// Library/POUs/ForceControl/MC_ReadActualForce/Structures/ReadActualForceSendData
{attribute 'pack_mode' := '1'}
// ------------------------------------------------------------------------- 
//  SRCI Robot Library                                                
// ------------------------------------------------------------------------- 
//                                                                           
//  Object:      ReadActualForceSendData                                       
//  Author:      Thorsten Brach                                                
//  Date:        2024-06-11
//
//  Description:                                              
//   
//                                                                           
//  Copyright: 
//    (C) 2024 Thorsten Brach. All rights reserved                                                                                                                                            
//             Licensed under the LGPL-3.0 license.
//                                                                           
//  Disclaimer:                                                                           
//    This project is provided without any guarantee and can be used for   
//    private and commercial purposes. Any use is at the user’s 
//    own risk and responsibility.
//
// -------------------------------------------------------------------------
TYPE ReadActualForceSendData EXTENDS CmdHeader:   
STRUCT
  /// ID of Action that will be executed when this command is active
  /// • >0: Start Action        - Start executing the Action function with the identical ListenerID.
  /// • <0: Stop Action         - Stop executing the Action function with the identical ListenerID.
  /// •  0: Undefined (default) - If no EmitterID is defined, the function returns an error message
  /// For more information see chapter 5.5.12.4
  EmitterID          : ARRAY [0..3] OF SINT;
  /// ListenerID
  ListenerID         : SINT; 
  /// Reserve
  Reserve            : BYTE; 
  /// Index of tool
  /// •      0: Flange (default)
  /// • 1..254: Tool frames
  ToolNo             : USINT;
  /// Define the index number of the UCS that will be assigned to the conveyor.
  /// For more information refer to chapter 5.5.14
  FrameNo            : USINT;
  /// Index of payload data containing mass, center of gravity, orientation and inertia relative to SensorFrame.
  /// Required to calibrate system for setting up gravity compensation and sensor offset.
  CalibrationData    : USINT;
  /// Defines type of reference of Force and Torque (at least one option must be supported )
  ReferenceType      : ReferenceType;
END_STRUCT
END_TYPE

// Library/POUs/General/MC_EnableRobot/Structures/EnableRobotOutCmd
{attribute 'pack_mode' := '1'} 
// ------------------------------------------------------------------------- 
//  SRCI Robot Library                                                
// ------------------------------------------------------------------------- 
//                                                                           
//  Object:      EnableRobotOutCmd                                       
//  Author:      Thorsten Brach                                                
//  Date:        2024-06-01
//
//  Description:                                              
//   
//                                                                           
//  Copyright: 
//    (C) 2024 Thorsten Brach. All rights reserved                                                                                                                                            
//             Licensed under the LGPL-3.0 license.
//                                                                           
//  Disclaimer:                                                                           
//    This project is provided without any guarantee and can be used for   
//    private and commercial purposes. Any use is at the user’s 
//    own risk and responsibility.
//
// -------------------------------------------------------------------------
TYPE EnableRobotOutCmd :
STRUCT
END_STRUCT
END_TYPE

// Library/POUs/General/MC_EnableRobot/Structures/EnableRobotParCmd
{attribute 'pack_mode' := '1'} 
// ------------------------------------------------------------------------- 
//  SRCI Robot Library                                                
// ------------------------------------------------------------------------- 
//                                                                           
//  Object:      EnableRobotParCmd                                       
//  Author:      Thorsten Brach                                                
//  Date:        2024-06-01
//
//  Description:                                              
//   
//                                                                           
//  Copyright: 
//    (C) 2024 Thorsten Brach. All rights reserved                                                                                                                                            
//             Licensed under the LGPL-3.0 license.
//                                                                           
//  Disclaimer:                                                                           
//    This project is provided without any guarantee and can be used for   
//    private and commercial purposes. Any use is at the user’s 
//    own risk and responsibility.
//
// -------------------------------------------------------------------------
TYPE EnableRobotParCmd :
STRUCT
  /// The robot will move while HoldToRun is set TRUE
  HoldToRun  : BOOL;
  /// While activated the RI state switches to interrupted when a buffered command returns Done TRUE
  /// At least one of the optional modes must be supported
  StepMode   : StepMode;
  /// Relates to StepMode 1 (Blending) and 2 (Exact stop)
  /// Start the next buffered command with the rising edge in T1 External or T2 External
  ManualStep : BOOL;  
END_STRUCT
END_TYPE

// Library/POUs/General/MC_EnableRobot/Structures/EnableRobotRecvData
{attribute 'pack_mode' := '1'} 
// ------------------------------------------------------------------------- 
//  SRCI Robot Library                                                
// ------------------------------------------------------------------------- 
//                                                                           
//  Object:      EnableRobotRecvData                                       
//  Author:      Thorsten Brach                                                
//  Date:        2024-06-01
//
//  Description:                                              
//   
//                                                                           
//  Copyright: 
//    (C) 2024 Thorsten Brach. All rights reserved                                                                                                                                            
//             Licensed under the LGPL-3.0 license.
//                                                                           
//  Disclaimer:                                                                           
//    This project is provided without any guarantee and can be used for   
//    private and commercial purposes. Any use is at the user’s 
//    own risk and responsibility.
//
// -------------------------------------------------------------------------
TYPE EnableRobotRecvData EXTENDS RspHeader :
STRUCT
  /// TRUE when robot is set to RA power state "Enabled".
  Enabled : BOOL;
END_STRUCT
END_TYPE

// Library/POUs/General/MC_EnableRobot/Structures/EnableRobotSendData
{attribute 'pack_mode' := '1'}
// ------------------------------------------------------------------------- 
//  SRCI Robot Library                                                
// ------------------------------------------------------------------------- 
//                                                                           
//  Object:      ActivateNextCommandParCmd                                       
//  Author:      Thorsten Brach                                                
//  Date:        2024-06-01
//
//  Description:                                              
//   
//                                                                           
//  Copyright: 
//    (C) 2024 Thorsten Brach. All rights reserved                                                                                                                                            
//             Licensed under the LGPL-3.0 license.
//                                                                           
//  Disclaimer:                                                                           
//    This project is provided without any guarantee and can be used for   
//    private and commercial purposes. Any use is at the user’s 
//    own risk and responsibility.
//
// -------------------------------------------------------------------------
TYPE EnableRobotSendData EXTENDS CmdHeader: 
STRUCT
  /// Set TRUE to change RA power state to "Enabled"
 Enable          : BOOL;
 /// The robot will move while HoldToRun is set TRUE
 HoldToRun       : BOOL;
 /// While activated the RI state switches to interrupted when a buffered command returns Done TRUE
 /// At least one of the optional modes must be supported
 StepMode        : StepMode;
 /// Relates to StepMode 1 (Blending) and 2 (Exact stop)
 /// Start the next buffered command with the rising edge in T1 External or T2 External
 ManualStep      : BOOL;  
END_STRUCT
END_TYPE

// Library/POUs/General/MC_GroupReset/Structures/GroupResetOutCmd
{attribute 'pack_mode' := '1'} 
// ------------------------------------------------------------------------- 
//  SRCI Robot Library                                                
// ------------------------------------------------------------------------- 
//                                                                           
//  Object:      GroupResetOutCmd                                       
//  Author:      Thorsten Brach                                                
//  Date:        2024-06-17
//
//  Description:                                              
//   
//                                                                           
//  Copyright: 
//    (C) 2024 Thorsten Brach. All rights reserved                                                                                                                                            
//             Licensed under the LGPL-3.0 license.
//                                                                           
//  Disclaimer:                                                                           
//    This project is provided without any guarantee and can be used for   
//    private and commercial purposes. Any use is at the user’s 
//    own risk and responsibility.
//
// -------------------------------------------------------------------------
TYPE GroupResetOutCmd :
STRUCT
END_STRUCT
END_TYPE

// Library/POUs/General/MC_GroupReset/Structures/GroupResetParCmd
{attribute 'pack_mode' := '1'} 
// ------------------------------------------------------------------------- 
//  SRCI Robot Library                                                
// ------------------------------------------------------------------------- 
//                                                                           
//  Object:      GroupResetParCmd                                       
//  Author:      Thorsten Brach                                                
//  Date:        2024-06-17
//
//  Description:                                              
//   
//                                                                           
//  Copyright: 
//    (C) 2024 Thorsten Brach. All rights reserved                                                                                                                                            
//             Licensed under the LGPL-3.0 license.
//                                                                           
//  Disclaimer:                                                                           
//    This project is provided without any guarantee and can be used for   
//    private and commercial purposes. Any use is at the user’s 
//    own risk and responsibility.
//
// -------------------------------------------------------------------------
TYPE GroupResetParCmd :
STRUCT
END_STRUCT
END_TYPE

// Library/POUs/General/MC_GroupReset/Structures/GroupResetRecvData
{attribute 'pack_mode' := '1'} 
// ------------------------------------------------------------------------- 
//  SRCI Robot Library                                                
// ------------------------------------------------------------------------- 
//                                                                           
//  Object:      GroupResetRecvData                                       
//  Author:      Thorsten Brach                                                
//  Date:        2024-06-17
//
//  Description:                                              
//   
//                                                                           
//  Copyright: 
//    (C) 2024 Thorsten Brach. All rights reserved                                                                                                                                            
//             Licensed under the LGPL-3.0 license.
//                                                                           
//  Disclaimer:                                                                           
//    This project is provided without any guarantee and can be used for   
//    private and commercial purposes. Any use is at the user’s 
//    own risk and responsibility.
//
// -------------------------------------------------------------------------
TYPE GroupResetRecvData EXTENDS RspHeader :
STRUCT
END_STRUCT
END_TYPE

// Library/POUs/General/MC_GroupReset/Structures/GroupResetSendData
{attribute 'pack_mode' := '1'}
// ------------------------------------------------------------------------- 
//  SRCI Robot Library                                                
// ------------------------------------------------------------------------- 
//                                                                           
//  Object:      GroupResetSendData                                       
//  Author:      Thorsten Brach                                                
//  Date:        2024-06-17
//
//  Description:                                              
//   
//                                                                           
//  Copyright: 
//    (C) 2024 Thorsten Brach. All rights reserved                                                                                                                                            
//             Licensed under the LGPL-3.0 license.
//                                                                           
//  Disclaimer:                                                                           
//    This project is provided without any guarantee and can be used for   
//    private and commercial purposes. Any use is at the user’s 
//    own risk and responsibility.
//
// -------------------------------------------------------------------------
TYPE GroupResetSendData EXTENDS CmdHeader:   
STRUCT
END_STRUCT
END_TYPE

// Library/POUs/General/MC_RestartController/Structures/RestartControllerOutCmd
{attribute 'pack_mode' := '1'} 
// ------------------------------------------------------------------------- 
//  SRCI Robot Library                                                
// ------------------------------------------------------------------------- 
//                                                                           
//  Object:      RestartControllerOutCmd                                       
//  Author:      Thorsten Brach                                                
//  Date:        2024-06-22
//
//  Description:                                              
//   
//                                                                           
//  Copyright: 
//    (C) 2024 Thorsten Brach. All rights reserved                                                                                                                                            
//             Licensed under the LGPL-3.0 license.
//                                                                           
//  Disclaimer:                                                                           
//    This project is provided without any guarantee and can be used for   
//    private and commercial purposes. Any use is at the user’s 
//    own risk and responsibility.
//
// -------------------------------------------------------------------------
TYPE RestartControllerOutCmd :
STRUCT
  /// TRUE when execution of command has been confirmed by RC and restart is about to be initiated.
  RestartAccepted : BOOL;  
END_STRUCT
END_TYPE

// Library/POUs/General/MC_RestartController/Structures/RestartControllerParCmd
{attribute 'pack_mode' := '1'} 
// ------------------------------------------------------------------------- 
//  SRCI Robot Library                                                
// ------------------------------------------------------------------------- 
//                                                                           
//  Object:      RestartControllerParCmd                                       
//  Author:      Thorsten Brach                                                
//  Date:        2024-06-22
//
//  Description:                                              
//   
//                                                                           
//  Copyright: 
//    (C) 2024 Thorsten Brach. All rights reserved                                                                                                                                            
//             Licensed under the LGPL-3.0 license.
//                                                                           
//  Disclaimer:                                                                           
//    This project is provided without any guarantee and can be used for   
//    private and commercial purposes. Any use is at the user’s 
//    own risk and responsibility.
//
// -------------------------------------------------------------------------
TYPE RestartControllerParCmd :
STRUCT
END_STRUCT
END_TYPE

// Library/POUs/General/MC_RestartController/Structures/RestartControllerRecvData
{attribute 'pack_mode' := '1'} 
// ------------------------------------------------------------------------- 
//  SRCI Robot Library                                                
// ------------------------------------------------------------------------- 
//                                                                           
//  Object:      RestartControllerRecvData                                       
//  Author:      Thorsten Brach                                                
//  Date:        2024-06-22
//
//  Description:                                              
//   
//                                                                           
//  Copyright: 
//    (C) 2024 Thorsten Brach. All rights reserved                                                                                                                                            
//             Licensed under the LGPL-3.0 license.
//                                                                           
//  Disclaimer:                                                                           
//    This project is provided without any guarantee and can be used for   
//    private and commercial purposes. Any use is at the user’s 
//    own risk and responsibility.
//
// -------------------------------------------------------------------------
TYPE RestartControllerRecvData EXTENDS RspHeader :
STRUCT
  /// TRUE when execution of command has been confirmed by RC and restart is about to be initiated.
  RestartAccepted : BOOL;
END_STRUCT
END_TYPE

// Library/POUs/General/MC_RestartController/Structures/RestartControllerSendData
{attribute 'pack_mode' := '1'}
// ------------------------------------------------------------------------- 
//  SRCI Robot Library                                                
// ------------------------------------------------------------------------- 
//                                                                           
//  Object:      RestartControllerSendData                                       
//  Author:      Thorsten Brach                                                
//  Date:        2024-06-22
//
//  Description:                                              
//   
//                                                                           
//  Copyright: 
//    (C) 2024 Thorsten Brach. All rights reserved                                                                                                                                            
//             Licensed under the LGPL-3.0 license.
//                                                                           
//  Disclaimer:                                                                           
//    This project is provided without any guarantee and can be used for   
//    private and commercial purposes. Any use is at the user’s 
//    own risk and responsibility.
//
// -------------------------------------------------------------------------
TYPE RestartControllerSendData EXTENDS CmdHeader: 
STRUCT
END_STRUCT
END_TYPE

// Library/POUs/General/MC_RobotTask/Structures/ParCfg/Com/RobotTaskParCfgCom
{attribute 'pack_mode' := '1'} 
// ------------------------------------------------------------------------- 
//  SRCI Robot Library                                                
// ------------------------------------------------------------------------- 
//                                                                           
//  Object:      RobotTaskParCfgCom                                       
//  Author:      Thorsten Brach                                                
//  Date:        2024-11-30
//
//  Description:                                              
//   
//                                                                           
//  Copyright: 
//    (C) 2024 Thorsten Brach. All rights reserved                                                                                                                                            
//             Licensed under the LGPL-3.0 license.
//                                                                           
//  Disclaimer:                                                                           
//    This project is provided without any guarantee and can be used for   
//    private and commercial purposes. Any use is at the user’s 
//    own risk and responsibility.
//
// -------------------------------------------------------------------------
TYPE RobotTaskParCfgCom :
STRUCT
  /// Maximum allowed time between incrementation of LifeSign before communication error.
  /// • <10 ms: Invalid
  /// • 50 ms: default
  /// See also chapter 5.6.6.2.
  LifeSignTimeOut        : TIME := T#50MS;
  /// Number of Bytes of the frame to be used for the telegram of the given Axisgroup. Direction client to server
  TelegramLengthPlcToRob : UINT := 256;
  /// Number of Bytes of the frame to be used for the telegram of the given Axisgroup. Direction server to client
  TelegramLengthRobToPlc : UINT := 256;  
END_STRUCT
END_TYPE

// Library/POUs/General/MC_RobotTask/Structures/ParCfg/Plc/RobotTaskParCfgPlc
{attribute 'pack_mode' := '1'} 
// ------------------------------------------------------------------------- 
//  SRCI Robot Library                                                
// ------------------------------------------------------------------------- 
//                                                                           
//  Object:      RobotTaskParCfgPlc                                       
//  Author:      Thorsten Brach                                                
//  Date:        2024-11-30
//
//  Description:                                              
//   
//                                                                           
//  Copyright: 
//    (C) 2024 Thorsten Brach. All rights reserved                                                                                                                                            
//             Licensed under the LGPL-3.0 license.
//                                                                           
//  Disclaimer:                                                                           
//    This project is provided without any guarantee and can be used for   
//    private and commercial purposes. Any use is at the user’s 
//    own risk and responsibility.
//
// -------------------------------------------------------------------------
TYPE RobotTaskParCfgPlc :
STRUCT
  /// PLC cycle time
  CycleTime           : TIME := T#10MS;
  /// parameter
  Parameter           : RobotTaskParCfgPlcParameter;  
  /// Configuration of optional cyclic data send to the Robot
  OptionalCyclic      : AxesGroupParameterPlcOptionalCyclic; {warning 'Remove - this is already part of RobotTaskParCfgPlcParameter'}
END_STRUCT
END_TYPE

// Library/POUs/General/MC_RobotTask/Structures/ParCfg/Plc/RobotTaskParCfgPlcParameter
{attribute 'pack_mode' := '1'} 
// ------------------------------------------------------------------------- 
//  SRCI Robot Library                                                
// ------------------------------------------------------------------------- 
//                                                                           
//  Object:      RobotTaskParCfgPlcParameter                                       
//  Author:      Thorsten Brach                                                
//  Date:        2024-11-30
//
//  Description:                                              
//   
//                                                                           
//  Copyright: 
//    (C) 2024 Thorsten Brach. All rights reserved                                                                                                                                            
//             Licensed under the LGPL-3.0 license.
//                                                                           
//  Disclaimer:                                                                           
//    This project is provided without any guarantee and can be used for   
//    private and commercial purposes. Any use is at the user’s 
//    own risk and responsibility.
//
// -------------------------------------------------------------------------
TYPE RobotTaskParCfgPlcParameter EXTENDS AxesGroupParameterPlcParameter :
STRUCT
END_STRUCT
END_TYPE

// Library/POUs/General/MC_RobotTask/Structures/ParCfg/Rob/RobotTaskParCfgRob
TYPE RobotTaskParCfgRob :
STRUCT
// ------------------------------------------------------------------------- 
//  SRCI Robot Library                                                
// ------------------------------------------------------------------------- 
//                                                                           
//  Object:      RobotTaskParCfgRob                                       
//  Author:      Thorsten Brach                                                
//  Date:        2024-11-30
//
//  Description:                                              
//   
//                                                                           
//  Copyright: 
//    (C) 2024 Thorsten Brach. All rights reserved                                                                                                                                            
//             Licensed under the LGPL-3.0 license.
//                                                                           
//  Disclaimer:                                                                           
//    This project is provided without any guarantee and can be used for   
//    private and commercial purposes. Any use is at the user’s 
//    own risk and responsibility.
//
// -------------------------------------------------------------------------
  /// Robot parameter
  Parameter      : RobotTaskParCfgRobParameter;
  /// Configuration of optional cyclic data received from the Robot
  OptionalCyclic : AxesGroupParameterRobOptionalCyclic;
END_STRUCT
END_TYPE

// Library/POUs/General/MC_RobotTask/Structures/ParCfg/Rob/RobotTaskParCfgRobParameter
{attribute 'pack_mode' := '1'} 
// ------------------------------------------------------------------------- 
//  SRCI Robot Library                                                
// ------------------------------------------------------------------------- 
//                                                                           
//  Object:      RobotTaskParCfgRobParameter                                       
//  Author:      Thorsten Brach                                                
//  Date:        2024-11-30
//
//  Description:                                              
//   
//                                                                           
//  Copyright: 
//    (C) 2024 Thorsten Brach. All rights reserved                                                                                                                                            
//             Licensed under the LGPL-3.0 license.
//                                                                           
//  Disclaimer:                                                                           
//    This project is provided without any guarantee and can be used for   
//    private and commercial purposes. Any use is at the user’s 
//    own risk and responsibility.
//
// -------------------------------------------------------------------------
TYPE RobotTaskParCfgRobParameter :
STRUCT
  /// Defines blending behavior for single move commands. One of the optional modes must be supported.
  ///  • 0 (default): Move to end position
  ///       Robot moves exactly the target position independently of the selected "BlendingMode"
  ///  • 1: Wait at blending parameter 
  ///       Robot stops its movement when the specified blending parameter is reached
  WaitAtBlendingZone         : BOOL;
  /// Allow a sequence switch from primary to secondary while a subprogram called via CallSubprogram (6.5.18) in the sequence is in progress
  AllowSecSeqWhileSubprogram : BOOL;
  /// Allows blending when CallSubprogram is called in sequence and removed afterwards. For more information see chapter 6.5.21.
  /// • 0 (default): Dynamic blending is prevented
  /// • 1: Dynamic blending is allowed
  AllowDynamicBlending       : BOOL;
  /// Defines waiting time of RC between receiving a first move command when motion queue is empty and starting the first movement. See also chapter 5.6.8.
  DelayTime                  : UINT;
  /// Define number of points required to calculate the blending. See also chapter 5.6.8.
  WaitForNrOfCmd             : UINT;
  /// Defines a delay time between detecting an inconsistency of configuration data between server and client and executing the defined SyncReaction. 
  /// Always positive. Default: 0 ms
  SyncDelay                  : UINT;
  /// Specifies system reaction in case inconsistency of synchronization data is detected according to Table 6-81. For more information refer to chapter 5.6.7.2
  SyncReaction               : SyncReaction;
  /// Enable datas to synchronize
  DataEnableSync             : DataEnableSync;
END_STRUCT
END_TYPE

// Library/POUs/General/MC_RobotTask/Structures/ParCfg/RobotTaskParCfg
{attribute 'pack_mode' := '1'} 
// ------------------------------------------------------------------------- 
//  SRCI Robot Library                                                
// ------------------------------------------------------------------------- 
//                                                                           
//  Object:      RobotTaskParCfg                                       
//  Author:      Thorsten Brach                                                
//  Date:        2024-11-30
//
//  Description:                                              
//   
//                                                                           
//  Copyright: 
//    (C) 2024 Thorsten Brach. All rights reserved                                                                                                                                            
//             Licensed under the LGPL-3.0 license.
//                                                                           
//  Disclaimer:                                                                           
//    This project is provided without any guarantee and can be used for   
//    private and commercial purposes. Any use is at the user’s 
//    own risk and responsibility.
//
// -------------------------------------------------------------------------
TYPE RobotTaskParCfg :
STRUCT
  /// Common parameter
  Com    : RobotTaskParCfgCom;
  /// PLC parameter
  Plc    : RobotTaskParCfgPlc;
  /// Robot parameter
  Rob    : RobotTaskParCfgRob; 
END_STRUCT
END_TYPE

// Library/POUs/General/MC_SetOperationMode/Structures/SetOperationModeOutCmd
{attribute 'pack_mode' := '1'} 
// ------------------------------------------------------------------------- 
//  SRCI Robot Library                                                
// ------------------------------------------------------------------------- 
//                                                                           
//  Object:      SetOperationModeOutCmd                                       
//  Author:      Thorsten Brach                                                
//  Date:        2024-08-01
//
//  Description:                                              
//   
//                                                                           
//  Copyright: 
//    (C) 2024 Thorsten Brach. All rights reserved                                                                                                                                            
//             Licensed under the LGPL-3.0 license.
//                                                                           
//  Disclaimer:                                                                           
//    This project is provided without any guarantee and can be used for   
//    private and commercial purposes. Any use is at the user’s 
//    own risk and responsibility.
//
// -------------------------------------------------------------------------
TYPE SetOperationModeOutCmd :
STRUCT
END_STRUCT
END_TYPE

// Library/POUs/General/MC_SetOperationMode/Structures/SetOperationModeParCmd
{attribute 'pack_mode' := '1'} 
// ------------------------------------------------------------------------- 
//  SRCI Robot Library                                                
// ------------------------------------------------------------------------- 
//                                                                           
//  Object:      SetOperationModeParCmd                                       
//  Author:      Thorsten Brach                                                
//  Date:        2024-08-01
//
//  Description:                                              
//   
//                                                                           
//  Copyright: 
//    (C) 2024 Thorsten Brach. All rights reserved                                                                                                                                            
//             Licensed under the LGPL-3.0 license.
//                                                                           
//  Disclaimer:                                                                           
//    This project is provided without any guarantee and can be used for   
//    private and commercial purposes. Any use is at the user’s 
//    own risk and responsibility.
//
// -------------------------------------------------------------------------
TYPE SetOperationModeParCmd :
STRUCT
  /// Limits for joints and external axes according to Table 6-180.
  OperationMode : OperationMode;
END_STRUCT
END_TYPE

// Library/POUs/General/MC_SetOperationMode/Structures/SetOperationModeRecvData
{attribute 'pack_mode' := '1'} 
// ------------------------------------------------------------------------- 
//  SRCI Robot Library                                                
// ------------------------------------------------------------------------- 
//                                                                           
//  Object:      SetOperationModeRecvData                                       
//  Author:      Thorsten Brach                                                
//  Date:        2024-08-01
//
//  Description:                                              
//   
//                                                                           
//  Copyright: 
//    (C) 2024 Thorsten Brach. All rights reserved                                                                                                                                            
//             Licensed under the LGPL-3.0 license.
//                                                                           
//  Disclaimer:                                                                           
//    This project is provided without any guarantee and can be used for   
//    private and commercial purposes. Any use is at the user’s 
//    own risk and responsibility.
//
// -------------------------------------------------------------------------
TYPE SetOperationModeRecvData EXTENDS RspHeader :
STRUCT
END_STRUCT
END_TYPE

// Library/POUs/General/MC_SetOperationMode/Structures/SetOperationModeSendData
{attribute 'pack_mode' := '1'}
// ------------------------------------------------------------------------- 
//  SRCI Robot Library                                                
// ------------------------------------------------------------------------- 
//                                                                           
//  Object:      SetOperationModeSendData                                       
//  Author:      Thorsten Brach                                                
//  Date:        2024-08-01
//
//  Description:                                              
//   
//                                                                           
//  Copyright: 
//    (C) 2024 Thorsten Brach. All rights reserved                                                                                                                                            
//             Licensed under the LGPL-3.0 license.
//                                                                           
//  Disclaimer:                                                                           
//    This project is provided without any guarantee and can be used for   
//    private and commercial purposes. Any use is at the user’s 
//    own risk and responsibility.
//
// -------------------------------------------------------------------------
TYPE SetOperationModeSendData EXTENDS CmdHeader: 
STRUCT
  /// Limits for joints and external axes according to Table 6-180.
  OperationMode : USINT;
END_STRUCT
END_TYPE

// Library/POUs/General/MC_SetSequence/Structures/SetSequenceOutCmd
{attribute 'pack_mode' := '1'} 
// ------------------------------------------------------------------------- 
//  SRCI Robot Library                                                
// ------------------------------------------------------------------------- 
//                                                                           
//  Object:      SetSequenceOutCmd                                       
//  Author:      Thorsten Brach                                                
//  Date:        2024-08-01
//
//  Description:                                              
//   
//                                                                           
//  Copyright: 
//    (C) 2024 Thorsten Brach. All rights reserved                                                                                                                                            
//             Licensed under the LGPL-3.0 license.
//                                                                           
//  Disclaimer:                                                                           
//    This project is provided without any guarantee and can be used for   
//    private and commercial purposes. Any use is at the user’s 
//    own risk and responsibility.
//
// -------------------------------------------------------------------------
TYPE SetSequenceOutCmd :
STRUCT

END_STRUCT
END_TYPE

// Library/POUs/General/MC_SetSequence/Structures/SetSequenceParCmd
{attribute 'pack_mode' := '1'} 
// ------------------------------------------------------------------------- 
//  SRCI Robot Library                                                
// ------------------------------------------------------------------------- 
//                                                                           
//  Object:      SetSequenceParCmd                                       
//  Author:      Thorsten Brach                                                
//  Date:        2024-08-01
//
//  Description:                                              
//   
//                                                                           
//  Copyright: 
//    (C) 2024 Thorsten Brach. All rights reserved                                                                                                                                            
//             Licensed under the LGPL-3.0 license.
//                                                                           
//  Disclaimer:                                                                           
//    This project is provided without any guarantee and can be used for   
//    private and commercial purposes. Any use is at the user’s 
//    own risk and responsibility.
//
// -------------------------------------------------------------------------
TYPE SetSequenceParCmd :
STRUCT
  /// Defines sequence to be activated when function is executed
  TargetSequence  : SequenceFlag;
END_STRUCT
END_TYPE

// Library/POUs/General/MC_SetSequence/Structures/SetSequenceRecvData
{attribute 'pack_mode' := '1'} 
// ------------------------------------------------------------------------- 
//  SRCI Robot Library                                                
// ------------------------------------------------------------------------- 
//                                                                           
//  Object:      SetSequenceRecvData                                       
//  Author:      Thorsten Brach                                                
//  Date:        2024-08-01
//
//  Description:                                              
//   
//                                                                           
//  Copyright: 
//    (C) 2024 Thorsten Brach. All rights reserved                                                                                                                                            
//             Licensed under the LGPL-3.0 license.
//                                                                           
//  Disclaimer:                                                                           
//    This project is provided without any guarantee and can be used for   
//    private and commercial purposes. Any use is at the user’s 
//    own risk and responsibility.
//
// -------------------------------------------------------------------------
TYPE SetSequenceRecvData EXTENDS RspHeader :
STRUCT

END_STRUCT
END_TYPE

// Library/POUs/General/MC_SetSequence/Structures/SetSequenceSendData
{attribute 'pack_mode' := '1'}
// ------------------------------------------------------------------------- 
//  SRCI Robot Library                                                
// ------------------------------------------------------------------------- 
//                                                                           
//  Object:      SetSequenceSendData                                       
//  Author:      Thorsten Brach                                                
//  Date:        2024-08-01
//
//  Description:                                              
//   
//                                                                           
//  Copyright: 
//    (C) 2024 Thorsten Brach. All rights reserved                                                                                                                                            
//             Licensed under the LGPL-3.0 license.
//                                                                           
//  Disclaimer:                                                                           
//    This project is provided without any guarantee and can be used for   
//    private and commercial purposes. Any use is at the user’s 
//    own risk and responsibility.
//
// -------------------------------------------------------------------------
TYPE SetSequenceSendData EXTENDS CmdHeader: 
STRUCT
  /// Defines sequence to be activated when function is executed
  TargetSequence  : USINT;
END_STRUCT
END_TYPE

// Library/POUs/General/MC_SwitchLanguage/Structures/SwitchLanguageOutCmd
{attribute 'pack_mode' := '1'} 
// ------------------------------------------------------------------------- 
//  SRCI Robot Library                                                
// ------------------------------------------------------------------------- 
//                                                                           
//  Object:      SwitchLanguageOutCmd                                       
//  Author:      Thorsten Brach                                                
//  Date:        2024-06-30
//
//  Description:                                              
//   
//                                                                           
//  Copyright: 
//    (C) 2024 Thorsten Brach. All rights reserved                                                                                                                                            
//             Licensed under the LGPL-3.0 license.
//                                                                           
//  Disclaimer:                                                                           
//    This project is provided without any guarantee and can be used for   
//    private and commercial purposes. Any use is at the user’s 
//    own risk and responsibility.
//
// -------------------------------------------------------------------------
TYPE SwitchLanguageOutCmd :
STRUCT
  /// Two letter code of actual language used at the original operating panel of the robot.
  ActualLanguageCode : STRING(2);  
END_STRUCT
END_TYPE

// Library/POUs/General/MC_SwitchLanguage/Structures/SwitchLanguageParCmd
{attribute 'pack_mode' := '1'} 
// ------------------------------------------------------------------------- 
//  SRCI Robot Library                                                
// ------------------------------------------------------------------------- 
//                                                                           
//  Object:      SwitchLanguageParCmd                                       
//  Author:      Thorsten Brach                                                
//  Date:        2024-06-30
//
//  Description:                                              
//   
//                                                                           
//  Copyright: 
//    (C) 2024 Thorsten Brach. All rights reserved                                                                                                                                            
//             Licensed under the LGPL-3.0 license.
//                                                                           
//  Disclaimer:                                                                           
//    This project is provided without any guarantee and can be used for   
//    private and commercial purposes. Any use is at the user’s 
//    own risk and responsibility.
//
// -------------------------------------------------------------------------
TYPE SwitchLanguageParCmd :
STRUCT
  /// Two letter code of language to be set at the original operating panel of the robot (default: EN)
  LanguageCode : STRING(2);  
END_STRUCT
END_TYPE

// Library/POUs/General/MC_SwitchLanguage/Structures/SwitchLanguageRecvData
{attribute 'pack_mode' := '1'} 
// ------------------------------------------------------------------------- 
//  SRCI Robot Library                                                
// ------------------------------------------------------------------------- 
//                                                                           
//  Object:      SwitchLanguageRecvData                                       
//  Author:      Thorsten Brach                                                
//  Date:        2024-06-30
//
//  Description:                                              
//   
//                                                                           
//  Copyright: 
//    (C) 2024 Thorsten Brach. All rights reserved                                                                                                                                            
//             Licensed under the LGPL-3.0 license.
//                                                                           
//  Disclaimer:                                                                           
//    This project is provided without any guarantee and can be used for   
//    private and commercial purposes. Any use is at the user’s 
//    own risk and responsibility.
//
// -------------------------------------------------------------------------
TYPE SwitchLanguageRecvData EXTENDS RspHeader :
STRUCT
  /// Two letter code of actual language used at the original operating panel of the robot.
  ActualLanguageCode : STRING(2);    
END_STRUCT
END_TYPE

// Library/POUs/General/MC_SwitchLanguage/Structures/SwitchLanguageSendData
{attribute 'pack_mode' := '1'}
// ------------------------------------------------------------------------- 
//  SRCI Robot Library                                                
// ------------------------------------------------------------------------- 
//                                                                           
//  Object:      SwitchLanguageSendData                                       
//  Author:      Thorsten Brach                                                
//  Date:        2024-06-30
//
//  Description:                                              
//   
//                                                                           
//  Copyright: 
//    (C) 2024 Thorsten Brach. All rights reserved                                                                                                                                            
//             Licensed under the LGPL-3.0 license.
//                                                                           
//  Disclaimer:                                                                           
//    This project is provided without any guarantee and can be used for   
//    private and commercial purposes. Any use is at the user’s 
//    own risk and responsibility.
//
// -------------------------------------------------------------------------
TYPE SwitchLanguageSendData EXTENDS CmdHeader: 
STRUCT
  /// Two letter code of language to be set at the original operating panel of the robot (default: EN)
  LanguageCode : STRING(2);    
END_STRUCT
END_TYPE

// Library/POUs/General/MC_UserLogin/Structures/UserLoginOutCmd
{attribute 'pack_mode' := '1'} 
// ------------------------------------------------------------------------- 
//  SRCI Robot Library                                                
// ------------------------------------------------------------------------- 
//                                                                           
//  Object:      UserLoginOutCmd                                       
//  Author:      Thorsten Brach                                                
//  Date:        2024-06-30
//
//  Description:                                              
//   
//                                                                           
//  Copyright: 
//    (C) 2024 Thorsten Brach. All rights reserved                                                                                                                                            
//             Licensed under the LGPL-3.0 license.
//                                                                           
//  Disclaimer:                                                                           
//    This project is provided without any guarantee and can be used for   
//    private and commercial purposes. Any use is at the user’s 
//    own risk and responsibility.
//
// -------------------------------------------------------------------------
TYPE UserLoginOutCmd :
STRUCT
END_STRUCT
END_TYPE

// Library/POUs/General/MC_UserLogin/Structures/UserLoginParCmd
{attribute 'pack_mode' := '1'} 
// ------------------------------------------------------------------------- 
//  SRCI Robot Library                                                
// ------------------------------------------------------------------------- 
//                                                                           
//  Object:      UserLoginParCmd                                       
//  Author:      Thorsten Brach                                                
//  Date:        2024-06-30
//
//  Description:                                              
//   
//                                                                           
//  Copyright: 
//    (C) 2024 Thorsten Brach. All rights reserved                                                                                                                                            
//             Licensed under the LGPL-3.0 license.
//                                                                           
//  Disclaimer:                                                                           
//    This project is provided without any guarantee and can be used for   
//    private and commercial purposes. Any use is at the user’s 
//    own risk and responsibility.
//
// -------------------------------------------------------------------------
TYPE UserLoginParCmd :
STRUCT
  /// Defines the logon type (at least one option must be supported)
  Mode            : LogonMode;
  /// Defines the user password.
  Password        : STRING(50);
  /// Defines the name of the operator
  Username        : STRING(50);
  /// Defines the level ID of the operator (default: 0)
  LevelID         : SINT;  
END_STRUCT
END_TYPE

// Library/POUs/General/MC_UserLogin/Structures/UserLoginRecvData
{attribute 'pack_mode' := '1'} 
// ------------------------------------------------------------------------- 
//  SRCI Robot Library                                                
// ------------------------------------------------------------------------- 
//                                                                           
//  Object:      UserLoginRecvData                                       
//  Author:      Thorsten Brach                                                
//  Date:        2024-06-30
//
//  Description:                                              
//   
//                                                                           
//  Copyright: 
//    (C) 2024 Thorsten Brach. All rights reserved                                                                                                                                            
//             Licensed under the LGPL-3.0 license.
//                                                                           
//  Disclaimer:                                                                           
//    This project is provided without any guarantee and can be used for   
//    private and commercial purposes. Any use is at the user’s 
//    own risk and responsibility.
//
// -------------------------------------------------------------------------
TYPE UserLoginRecvData EXTENDS RspHeader :
STRUCT
END_STRUCT
END_TYPE

// Library/POUs/General/MC_UserLogin/Structures/UserLoginSendData
{attribute 'pack_mode' := '1'}
// ------------------------------------------------------------------------- 
//  SRCI Robot Library                                                
// ------------------------------------------------------------------------- 
//                                                                           
//  Object:      UserLoginSendData                                       
//  Author:      Thorsten Brach                                                
//  Date:        2024-06-30
//
//  Description:                                              
//   
//                                                                           
//  Copyright: 
//    (C) 2024 Thorsten Brach. All rights reserved                                                                                                                                            
//             Licensed under the LGPL-3.0 license.
//                                                                           
//  Disclaimer:                                                                           
//    This project is provided without any guarantee and can be used for   
//    private and commercial purposes. Any use is at the user’s 
//    own risk and responsibility.
//
// -------------------------------------------------------------------------
TYPE UserLoginSendData EXTENDS CmdHeader: 
STRUCT
  /// Defines the logon type (at least one option must be supported)
  Mode            : LogonMode;
  /// Defines the level ID of the operator (default: 0)
  LevelID         : SINT;  
  /// Defines the user password.
  Password        : STRING(50);
  /// Defines the name of the operator
  Username        : STRING(50);
END_STRUCT
END_TYPE

// Library/POUs/Read/MC_ReadActualPosition/Structures/ReadActualPositionOutCmd
{attribute 'pack_mode' := '1'} 
// ------------------------------------------------------------------------- 
//  SRCI Robot Library                                                
// ------------------------------------------------------------------------- 
//                                                                           
//  Object:      ReadActualPositionOutCmd                                       
//  Author:      Thorsten Brach                                                
//  Date:        2024-08-09
//
//  Description:                                              
//   
//                                                                           
//  Copyright: 
//    (C) 2024 Thorsten Brach. All rights reserved                                                                                                                                            
//             Licensed under the LGPL-3.0 license.
//                                                                           
//  Disclaimer:                                                                           
//    This project is provided without any guarantee and can be used for   
//    private and commercial purposes. Any use is at the user’s 
//    own risk and responsibility.
//
// -------------------------------------------------------------------------
TYPE ReadActualPositionOutCmd :
STRUCT
  /// Relates to ListenerID >0 
  /// Number of successful trigger -based command invocations
  /// For more information refer to chapter 5.5.12.4.
  InvocationCounter       : USINT;
  /// Unique system-generated ID of the "Action" when the function is triggered.
  /// • >0: The "Action" is started by the trigger funcrion with identical FollowID.
  /// • <0: The "Action" is stopped by the trigger function with identical FollowID.
  /// For more information see chapter 5.5.12.4 EmitterID, ListenerID, FollowID and OriginID
  OriginID                : INT;
  /// Index of tool of returned position
  /// •     -1: Currently used tool on RC
  /// •      0: Flange (default)
  /// • 1..254: Tool frames
  ToolNoReturn            : INT;
  /// Index of frame of returned position
  /// •     -1: Currently used frame on RC
  /// •      0: WCS (default)
  /// • 1..254: User frames
  FrameNoReturn           : INT;
  /// Absolute coordinates in the active coordinate system
  ActualCartesianPosition : RobotCartesianPosition;
  /// Absolute position of the robot in Joint position.
  ActualJointPosition     : RobotJointPosition;
END_STRUCT
END_TYPE

// Library/POUs/Read/MC_ReadActualPosition/Structures/ReadActualPositionParCmd
{attribute 'pack_mode' := '1'} 
// ------------------------------------------------------------------------- 
//  SRCI Robot Library                                                
// ------------------------------------------------------------------------- 
//                                                                           
//  Object:      ReadActualPositionParCmd                                       
//  Author:      Thorsten Brach                                                
//  Date:        2024-08-09
//
//  Description:                                              
//   
//                                                                           
//  Copyright: 
//    (C) 2024 Thorsten Brach. All rights reserved                                                                                                                                            
//             Licensed under the LGPL-3.0 license.
//                                                                           
//  Disclaimer:                                                                           
//    This project is provided without any guarantee and can be used for   
//    private and commercial purposes. Any use is at the user’s 
//    own risk and responsibility.
//
// -------------------------------------------------------------------------
TYPE ReadActualPositionParCmd :
STRUCT
  /// Index of tool of returned position
  /// •     -1: Currently used tool on RC
  /// •      0: Flange (default)
  /// • 1..254: Tool frames
  ToolNo             : INT;
  /// Index of frame of returned position
  /// •     -1: Currently used frame on RC
  /// •      0: WCS (default)
  /// • 1..254: User frames
  FrameNo            : INT;
  /// ID of associated trigger function
  /// •  0: No Trigger (default) -> No trigger related behavior
  /// • >0: Trigger              -> Start executing when the trigger function with the identical EmitterID is triggered.
  /// Always positive. For more information, see chapter 5.5.12 Triggers
  ListenerID         : SINT;
END_STRUCT
END_TYPE

// Library/POUs/Read/MC_ReadActualPosition/Structures/ReadActualPositionRecvData
{attribute 'pack_mode' := '1'} 
// ------------------------------------------------------------------------- 
//  SRCI Robot Library                                                
// ------------------------------------------------------------------------- 
//                                                                           
//  Object:      ReadActualPositionRecvData                                       
//  Author:      Thorsten Brach                                                
//  Date:        2024-08-09
//
//  Description:                                              
//   
//                                                                           
//  Copyright: 
//    (C) 2024 Thorsten Brach. All rights reserved                                                                                                                                            
//             Licensed under the LGPL-3.0 license.
//                                                                           
//  Disclaimer:                                                                           
//    This project is provided without any guarantee and can be used for   
//    private and commercial purposes. Any use is at the user’s 
//    own risk and responsibility.
//
// -------------------------------------------------------------------------
TYPE ReadActualPositionRecvData EXTENDS RspHeader :
STRUCT
  /// Relates to ListenerID >0
  /// Number of successful trigger-based command invocations - For more information refer TO chapter 5.5.12.4
  InvocationCounter       : USINT;  
  /// Reserve
  Reserve                 : SINT;
  /// Unique system-generated ID of the "Action" when the function is triggered.
  /// • >0: The "Action" is started by the trigger funcrion with identical FollowID.
  /// • <0: The "Action" is stopped by the trigger function with identical FollowID.
  /// For more information see chapter 5.5.12.4 EmitterID, ListenerID, FollowID and OriginID
  OriginID                : INT;
  /// Index of tool of returned position
  /// •     -1: Currently used tool on RC
  /// •      0: Flange (default)
  /// • 1..254: Tool frames
  ToolNoReturn            : INT;
  /// Index of frame of returned position
  /// •     -1: Currently used frame on RC
  /// •      0: WCS (default)
  /// • 1..254: User frames
  FrameNoReturn           : INT;
  /// Absolute coordinates in the active coordinate system
  ActualCartesianPosition : RobotCartesianPosition;
  /// Absolute position of the robot in Joint position.
  ActualJointPosition     : RobotJointPosition;
END_STRUCT
END_TYPE

// Library/POUs/Read/MC_ReadActualPosition/Structures/ReadActualPositionSendData
{attribute 'pack_mode' := '1'}
// ------------------------------------------------------------------------- 
//  SRCI Robot Library                                                
// ------------------------------------------------------------------------- 
//                                                                           
//  Object:      ReadActualPositionSendData                                       
//  Author:      Thorsten Brach                                                
//  Date:        2024-08-09
//
//  Description:                                              
//   
//                                                                           
//  Copyright: 
//    (C) 2024 Thorsten Brach. All rights reserved                                                                                                                                            
//             Licensed under the LGPL-3.0 license.
//                                                                           
//  Disclaimer:                                                                           
//    This project is provided without any guarantee and can be used for   
//    private and commercial purposes. Any use is at the user’s 
//    own risk and responsibility.
//
// -------------------------------------------------------------------------
TYPE ReadActualPositionSendData EXTENDS CmdHeader: 
STRUCT
  /// ID of Action that will be executed when this command is active
  /// • >0: Start Action - Start executing the Action function with the identical ListenerID.
  /// • <0: Stop Action  -  Stop executing the Action function with the identical ListenerID.
  /// • 0: No trigger (default)-  If no EmitterID is defined, the function will not trigger any Action during its execution
  /// For more information see section Triggers of this chapter or chapter 5.5.12.4.
  EmitterID          : ARRAY [0..3] OF SINT;
  /// ID of associated trigger function:
  /// •  0: No Trigger (default)  No trigger related behavior
  /// • >0: Trigger - Start executing when the trigger function with the identical EmitterID is triggered.
  /// Always positive.
  /// For more information, see chapter 5.5.12 Triggers
  ListenerID         : SINT;
  /// Reserve
  Reserve            : BYTE;
  /// Index of tool of returned position
  /// •     -1: Currently used tool on RC
  /// •      0: Flange (default)
  /// • 1..254: Tool frames
  ToolNo             : USINT;
  /// Index of frame of returned position
  /// •     -1: Currently used frame on RC
  /// •      0: WCS (default)
  /// • 1..254: User frames
  FrameNo            : USINT;
END_STRUCT
END_TYPE

// Library/POUs/Read/MC_ReadActualPositionCyclic/Structures/ReadActualPositionCyclicOutCmd
{attribute 'pack_mode' := '1'} 
// ------------------------------------------------------------------------- 
//  SRCI Robot Library                                                
// ------------------------------------------------------------------------- 
//                                                                           
//  Object:      ReadActualPositionCyclicOutCmd                                       
//  Author:      Thorsten Brach                                                
//  Date:        2024-08-09
//
//  Description:                                              
//   
//                                                                           
//  Copyright: 
//    (C) 2024 Thorsten Brach. All rights reserved                                                                                                                                            
//             Licensed under the LGPL-3.0 license.
//                                                                           
//  Disclaimer:                                                                           
//    This project is provided without any guarantee and can be used for   
//    private and commercial purposes. Any use is at the user’s 
//    own risk and responsibility.
//
// -------------------------------------------------------------------------
TYPE ReadActualPositionCyclicOutCmd :
STRUCT
  /// TRUE, while the output CartesianPosition returns valid values
  ReadingCartesianPosition    : BOOL;
  /// TRUE, while the output ExtCartesianPosition returns valid values
  ReadingCartesianPositionExt : BOOL;
  /// TRUE, while the output JointPosition returns valid values
  ReadingJointPosition        : BOOL;
  /// TRUE, while the output ExtJointPosition returns valid values
  ReadingJointPositionExt     : BOOL;
  /// Tool and frame index of currently used tool and frame according to Table 6-40
  CurrentCoordinateSystem     : CoordinateSystem;
  /// Cyclically returned, absolute coordinates of current position in selected coordinate systems (see input parameters ToolNo and FrameNo) 
  CartesianPosition           : RobotCartesianPosition;
  /// Cyclically returned, absolute coordinates of current position in selected coordinate systems (see input parameters ToolNo and FrameNo) 
  CartesianPositionShort      : RobotCartesianPositionShort;
  /// Cyclically returned, absolute cartesian position of the external axes of the robot
  CartesianPositionExt        : RobotCartesianPositionExt;
  /// Tool and frame index of returned position according to Table 6-40
  CoordinateSystem            : CoordinateSystem;
  /// Cyclically returned, absolute joint position of the robot in Joint position
  JointPosition               : RobotJointPosition;
  /// Cyclically returned, absolute short joint position of the robot in Joint position
  JointPositionShort          : RobotJointPositionShort;
  /// Cyclically returned, absolute extended joint position of the external axes of the robot
  JointPositionExt            : RobotJointPositionExt;
END_STRUCT
END_TYPE

// Library/POUs/Read/MC_ReadActualPositionCyclic/Structures/ReadActualPositionCyclicParCmd
{attribute 'pack_mode' := '1'} 
// ------------------------------------------------------------------------- 
//  SRCI Robot Library                                                
// ------------------------------------------------------------------------- 
//                                                                           
//  Object:      ReadActualPositionCyclicParCmd                                       
//  Author:      Thorsten Brach                                                
//  Date:        2024-08-09
//
//  Description:                                              
//   
//                                                                           
//  Copyright: 
//    (C) 2024 Thorsten Brach. All rights reserved                                                                                                                                            
//             Licensed under the LGPL-3.0 license.
//                                                                           
//  Disclaimer:                                                                           
//    This project is provided without any guarantee and can be used for   
//    private and commercial purposes. Any use is at the user’s 
//    own risk and responsibility.
//
// -------------------------------------------------------------------------
TYPE ReadActualPositionCyclicParCmd :
STRUCT
  /// Set TRUE (default) to activate cyclic transmission of cartesian position without external axes
  ReadCartesianPosition       : BOOL;
  /// Set TRUE to activate cyclic transmission of external axes values of cartesian position -  Default: False
  ReadCartesianPositionExt    : BOOL;
  ///Index of tool of returned position
  /// •     -1: Currently used tool on RC
  /// •      0: Flange (default)
  /// • 1..254: Tool frames
  ToolNo                      : INT;
  /// Index of frame of returned position
  /// •     -1: Currently used frame on RC
  /// •      0: WCS (default)
  /// • 1..254: User frames
  FrameNo                     : INT;
  /// Set TRUE (default) to activate cyclic transmission of joint position without external axes
  ReadJointPosition           : BOOL;
  /// Set TRUE to activate cyclic transmission of external axes values of joint position - Default: False
  ReadJointPositionExt        : BOOL;
END_STRUCT
END_TYPE

// Library/POUs/Read/MC_ReadActualTCPVelocity/Structures/ReadActualTCPVelocityOutCmd
{attribute 'pack_mode' := '1'} 
// ------------------------------------------------------------------------- 
//  SRCI Robot Library                                                
// ------------------------------------------------------------------------- 
//                                                                           
//  Object:      ReadActualTCPVelocityOutCmd                                       
//  Author:      Thorsten Brach                                                
//  Date:        2024-08-09
//
//  Description:                                              
//   
//                                                                           
//  Copyright: 
//    (C) 2024 Thorsten Brach. All rights reserved                                                                                                                                            
//             Licensed under the LGPL-3.0 license.
//                                                                           
//  Disclaimer:                                                                           
//    This project is provided without any guarantee and can be used for   
//    private and commercial purposes. Any use is at the user’s 
//    own risk and responsibility.
//
// -------------------------------------------------------------------------
TYPE ReadActualTCPVelocityOutCmd :
STRUCT
  /// Absolute actual velocity of the robot’s TCP. [mm/s]
  ActualTCPVelocity  : REAL;
  /// Index of tool of returned velocity
  /// •      0: Flange
  /// • 1..254: Tool frames
  ToolNoReturn       : USINT;
  /// Index of frame of returned position
  /// •      0: WCS
  /// • 1..254: User frames
  FrameNoReturn      : USINT;
  /// Unique system-generated ID of the "Action" when the function is triggered
  /// • >0: The "Action" is started by the trigger function with identical FollowID.
  /// • <0: The "Action" is stopped by the trigger function with identical FollowID.
  /// For more information see chapter 5.5.12.4
  OriginID           : INT;
  /// Relates to ListenerID >0 Number of successful trigger -based command invocations 
  /// For more information refer to chapter 5.5.12.4
  InvocationCounter  : USINT;
END_STRUCT
END_TYPE

// Library/POUs/Read/MC_ReadActualTCPVelocity/Structures/ReadActualTCPVelocityParCmd
{attribute 'pack_mode' := '1'} 
// ------------------------------------------------------------------------- 
//  SRCI Robot Library                                                
// ------------------------------------------------------------------------- 
//                                                                           
//  Object:      ReadActualTCPVelocityParCmd                                       
//  Author:      Thorsten Brach                                                
//  Date:        2024-08-09
//
//  Description:                                              
//   
//                                                                           
//  Copyright: 
//    (C) 2024 Thorsten Brach. All rights reserved                                                                                                                                            
//             Licensed under the LGPL-3.0 license.
//                                                                           
//  Disclaimer:                                                                           
//    This project is provided without any guarantee and can be used for   
//    private and commercial purposes. Any use is at the user’s 
//    own risk and responsibility.
//
// -------------------------------------------------------------------------
TYPE ReadActualTCPVelocityParCmd :
STRUCT
  /// Index of tool of returned velocity
  /// •      0: Flange (default)
  /// • 1..254: Tool frames
  ToolNo             : USINT;
  /// Index of frame
  /// •      0: WCS (default)
  /// • 1..254: User frames
  FrameNo            : USINT;
END_STRUCT
END_TYPE

// Library/POUs/Read/MC_ReadActualTCPVelocity/Structures/ReadActualTCPVelocityRecvData
{attribute 'pack_mode' := '1'} 
// ------------------------------------------------------------------------- 
//  SRCI Robot Library                                                
// ------------------------------------------------------------------------- 
//                                                                           
//  Object:      ReadActualTCPVelocityRecvData                                       
//  Author:      Thorsten Brach                                                
//  Date:        2024-08-09
//
//  Description:                                              
//   
//                                                                           
//  Copyright: 
//    (C) 2024 Thorsten Brach. All rights reserved                                                                                                                                            
//             Licensed under the LGPL-3.0 license.
//                                                                           
//  Disclaimer:                                                                           
//    This project is provided without any guarantee and can be used for   
//    private and commercial purposes. Any use is at the user’s 
//    own risk and responsibility.
//
// -------------------------------------------------------------------------
TYPE ReadActualTCPVelocityRecvData EXTENDS RspHeader :
STRUCT
  /// Relates to ListenerID >0
  /// Number of successful trigger-based command invocations - For more information refer TO chapter 5.5.12.4
  InvocationCounter : USINT;  
  /// Reserve
  Reserve           : SINT;
  /// Unique system-generated ID of the "Action" when the function is triggered.
  /// • >0: The "Action" is started by the trigger funcrion with identical FollowID.
  /// • <0: The "Action" is stopped by the trigger function with identical FollowID.
  /// For more information see chapter 5.5.12.4 EmitterID, ListenerID, FollowID and OriginID
  OriginID          : INT;
  /// Absolute actual velocity of the robot’s TCP. [mm/s]
  ActualTCPVelocity  : REAL;
  /// Index of tool of returned velocity
  /// •      0: Flange
  /// • 1..254: Tool frames
  ToolNoReturn       : USINT;
  /// Index of frame of returned position
  /// •      0: WCS
  /// • 1..254: User frames
  FrameNoReturn      : USINT;  
END_STRUCT
END_TYPE

// Library/POUs/Read/MC_ReadActualTCPVelocity/Structures/ReadActualTCPVelocitySendData
{attribute 'pack_mode' := '1'}
// ------------------------------------------------------------------------- 
//  SRCI Robot Library                                                
// ------------------------------------------------------------------------- 
//                                                                           
//  Object:      ReadActualTCPVelocitySendData                                       
//  Author:      Thorsten Brach                                                
//  Date:        2024-08-09
//
//  Description:                                              
//   
//                                                                           
//  Copyright: 
//    (C) 2024 Thorsten Brach. All rights reserved                                                                                                                                            
//             Licensed under the LGPL-3.0 license.
//                                                                           
//  Disclaimer:                                                                           
//    This project is provided without any guarantee and can be used for   
//    private and commercial purposes. Any use is at the user’s 
//    own risk and responsibility.
//
// -------------------------------------------------------------------------
TYPE ReadActualTCPVelocitySendData EXTENDS CmdHeader: 
STRUCT
  /// Index of tool of returned velocity
  /// •      0: Flange (default)
  /// • 1..254: Tool frames
  ToolNo             : USINT;
  /// Index of frame
  /// •      0: WCS (default)
  /// • 1..254: User frames
  FrameNo            : USINT;
END_STRUCT
END_TYPE

// Library/POUs/Read/MC_ReadAnalogInput/Structures/ReadAnalogInputOutCmd
{attribute 'pack_mode' := '1'} 
// ------------------------------------------------------------------------- 
//  SRCI Robot Library                                                
// ------------------------------------------------------------------------- 
//                                                                           
//  Object:      ReadAnalogInputOutCmd                                       
//  Author:      Thorsten Brach                                                
//  Date:        2024-08-09
//
//  Description:                                              
//   
//                                                                           
//  Copyright: 
//    (C) 2024 Thorsten Brach. All rights reserved                                                                                                                                            
//             Licensed under the LGPL-3.0 license.
//                                                                           
//  Disclaimer:                                                                           
//    This project is provided without any guarantee and can be used for   
//    private and commercial purposes. Any use is at the user’s 
//    own risk and responsibility.
//
// -------------------------------------------------------------------------
TYPE ReadAnalogInputOutCmd :
STRUCT
  /// Relates to ListenerID >0 
  /// Number of successful trigger -based command invocations
  /// For more information refer to chapter 5.5.12.4.
  InvocationCounter  : USINT;
  /// Unique system-generated ID of the "Action" when the function is triggered.
  /// • >0: The "Action" is started by the trigger funcrion with identical FollowID.
  /// • <0: The "Action" is stopped by the trigger function with identical FollowID.
  /// For more information see chapter 5.5.12.4 EmitterID, ListenerID, FollowID and OriginID
  OriginID           : INT;
  /// Returned values of digital inputs
  /// Returned values of digital inputs
  /// Unit of returned Value
  Unit               : UnitType;
  /// Returned value of analog input
  Value              : REAL;
END_STRUCT
END_TYPE

// Library/POUs/Read/MC_ReadAnalogInput/Structures/ReadAnalogInputParCmd
{attribute 'pack_mode' := '1'} 
// ------------------------------------------------------------------------- 
//  SRCI Robot Library                                                
// ------------------------------------------------------------------------- 
//                                                                           
//  Object:      ReadAnalogInputParCmd                                       
//  Author:      Thorsten Brach                                                
//  Date:        2024-08-09
//
//  Description:                                              
//   
//                                                                           
//  Copyright: 
//    (C) 2024 Thorsten Brach. All rights reserved                                                                                                                                            
//             Licensed under the LGPL-3.0 license.
//                                                                           
//  Disclaimer:                                                                           
//    This project is provided without any guarantee and can be used for   
//    private and commercial purposes. Any use is at the user’s 
//    own risk and responsibility.
//
// -------------------------------------------------------------------------
TYPE ReadAnalogInputParCmd :
STRUCT
  /// Number of the analog input 1..32
  Index              : USINT; 
  /// ID of associated trigger function:
  /// •  0: No Trigger (default)  No trigger related behavior
  /// • >0: Trigger - Start executing when the trigger function with the identical EmitterID is triggered.
  /// Always positive.
  /// For more information, see chapter 5.5.12 Triggers
  ListenerID         : SINT;
END_STRUCT
END_TYPE

// Library/POUs/Read/MC_ReadAnalogInput/Structures/ReadAnalogInputRecvData
{attribute 'pack_mode' := '1'} 
// ------------------------------------------------------------------------- 
//  SRCI Robot Library                                                
// ------------------------------------------------------------------------- 
//                                                                           
//  Object:      ReadAnalogInputRecvData                                       
//  Author:      Thorsten Brach                                                
//  Date:        2024-08-09
//
//  Description:                                              
//   
//                                                                           
//  Copyright: 
//    (C) 2024 Thorsten Brach. All rights reserved                                                                                                                                            
//             Licensed under the LGPL-3.0 license.
//                                                                           
//  Disclaimer:                                                                           
//    This project is provided without any guarantee and can be used for   
//    private and commercial purposes. Any use is at the user’s 
//    own risk and responsibility.
//
// -------------------------------------------------------------------------
TYPE ReadAnalogInputRecvData EXTENDS RspHeader :
STRUCT
  /// Relates to ListenerID >0
  /// Number of successful trigger-based command invocations - For more information refer TO chapter 5.5.12.4
  InvocationCounter : USINT;  
  /// Reserve
  Reserve           : SINT;
  /// Unique system-generated ID of the "Action" when the function is triggered.
  /// • >0: The "Action" is started by the trigger funcrion with identical FollowID.
  /// • <0: The "Action" is stopped by the trigger function with identical FollowID.
  /// For more information see chapter 5.5.12.4 EmitterID, ListenerID, FollowID and OriginID
  OriginID          : INT;
  /// Returned values of digital inputs
  /// Returned values of digital inputs
  /// Unit of returned Value
  Unit               : USINT;
  /// Returned value of analog input
  Value              : REAL;  
END_STRUCT
END_TYPE

// Library/POUs/Read/MC_ReadAnalogInput/Structures/ReadAnalogInputSendData
{attribute 'pack_mode' := '1'}
// ------------------------------------------------------------------------- 
//  SRCI Robot Library                                                
// ------------------------------------------------------------------------- 
//                                                                           
//  Object:      ReadAnalogInputSendData                                       
//  Author:      Thorsten Brach                                                
//  Date:        2024-08-09
//
//  Description:                                              
//   
//                                                                           
//  Copyright: 
//    (C) 2024 Thorsten Brach. All rights reserved                                                                                                                                            
//             Licensed under the LGPL-3.0 license.
//                                                                           
//  Disclaimer:                                                                           
//    This project is provided without any guarantee and can be used for   
//    private and commercial purposes. Any use is at the user’s 
//    own risk and responsibility.
//
// -------------------------------------------------------------------------
TYPE ReadAnalogInputSendData EXTENDS CmdHeader: 
STRUCT
  /// ID of Action that will be executed when this command is active
  /// • >0: Start Action - Start executing the Action function with the identical ListenerID.
  /// • <0: Stop Action  -  Stop executing the Action function with the identical ListenerID.
  /// • 0: No trigger (default)-  If no EmitterID is defined, the function will not trigger any Action during its execution
  /// For more information see section Triggers of this chapter or chapter 5.5.12.4.
  EmitterID          : ARRAY [0..3] OF SINT;
  /// ID of associated trigger function:
  /// •  0: No Trigger (default)  No trigger related behavior
  /// • >0: Trigger - Start executing when the trigger function with the identical EmitterID is triggered.
  /// Always positive.
  /// For more information, see chapter 5.5.12 Triggers
  ListenerID         : SINT;
  /// Reserve
  Reserve            : BYTE;
  /// Number of the analog input 1..32
  Index              : USINT; 
END_STRUCT
END_TYPE

// Library/POUs/Read/MC_ReadDHParameter/Structures/ReadDHParameterOutCmd
{attribute 'pack_mode' := '1'} 
// ------------------------------------------------------------------------- 
//  SRCI Robot Library                                                
// ------------------------------------------------------------------------- 
//                                                                           
//  Object:      ReadDigitalInputsOutCmd                                       
//  Author:      Thorsten Brach                                                
//  Date:        2024-08-09
//
//  Description:                                              
//   
//                                                                           
//  Copyright: 
//    (C) 2024 Thorsten Brach. All rights reserved                                                                                                                                            
//             Licensed under the LGPL-3.0 license.
//                                                                           
//  Disclaimer:                                                                           
//    This project is provided without any guarantee and can be used for   
//    private and commercial purposes. Any use is at the user’s 
//    own risk and responsibility.
//
// -------------------------------------------------------------------------
TYPE ReadDHParameterOutCmd :
STRUCT
  /// Denavit–Hartenberg parameter
  DHParameter : DHParameter;
END_STRUCT
END_TYPE

// Library/POUs/Read/MC_ReadDHParameter/Structures/ReadDHParameterParCmd
{attribute 'pack_mode' := '1'} 
// ------------------------------------------------------------------------- 
//  SRCI Robot Library                                                
// ------------------------------------------------------------------------- 
//                                                                           
//  Object:      ReadDigitalInputsParCmd                                       
//  Author:      Thorsten Brach                                                
//  Date:        2024-08-09
//
//  Description:                                              
//   
//                                                                           
//  Copyright: 
//    (C) 2024 Thorsten Brach. All rights reserved                                                                                                                                            
//             Licensed under the LGPL-3.0 license.
//                                                                           
//  Disclaimer:                                                                           
//    This project is provided without any guarantee and can be used for   
//    private and commercial purposes. Any use is at the user’s 
//    own risk and responsibility.
//
// -------------------------------------------------------------------------
TYPE ReadDHParameterParCmd :
STRUCT
  /// Determines if returned DH parameters use modified convention or classic convention.
  /// • 0: Classic convention (default)
  /// • 1: Modified convention
  ModifiedConvention : BOOL;  
END_STRUCT
END_TYPE

// Library/POUs/Read/MC_ReadDHParameter/Structures/ReadDHParameterRecvData
{attribute 'pack_mode' := '1'} 
// ------------------------------------------------------------------------- 
//  SRCI Robot Library                                                
// ------------------------------------------------------------------------- 
//                                                                           
//  Object:      ReadDigitalInputsRecvData                                       
//  Author:      Thorsten Brach                                                
//  Date:        2024-08-09
//
//  Description:                                              
//   
//                                                                           
//  Copyright: 
//    (C) 2024 Thorsten Brach. All rights reserved                                                                                                                                            
//             Licensed under the LGPL-3.0 license.
//                                                                           
//  Disclaimer:                                                                           
//    This project is provided without any guarantee and can be used for   
//    private and commercial purposes. Any use is at the user’s 
//    own risk and responsibility.
//
// -------------------------------------------------------------------------
TYPE ReadDHParameterRecvData EXTENDS RspHeader :
STRUCT
  /// Denavit–Hartenberg parameter
  DHParameter : DHParameter;  
END_STRUCT
END_TYPE

// Library/POUs/Read/MC_ReadDHParameter/Structures/ReadDHParameterSendData
{attribute 'pack_mode' := '1'}
// ------------------------------------------------------------------------- 
//  SRCI Robot Library                                                
// ------------------------------------------------------------------------- 
//                                                                           
//  Object:      ReadDigitalInputsSendData                                       
//  Author:      Thorsten Brach                                                
//  Date:        2024-08-09
//
//  Description:                                              
//   
//                                                                           
//  Copyright: 
//    (C) 2024 Thorsten Brach. All rights reserved                                                                                                                                            
//             Licensed under the LGPL-3.0 license.
//                                                                           
//  Disclaimer:                                                                           
//    This project is provided without any guarantee and can be used for   
//    private and commercial purposes. Any use is at the user’s 
//    own risk and responsibility.
//
// -------------------------------------------------------------------------
TYPE ReadDHParameterSendData EXTENDS CmdHeader: 
STRUCT
  /// Determines if returned DH parameters use modified convention or classic convention.
  /// • 0: Classic convention (default)
  /// • 1: Modified convention
  ModifiedConvention : BOOL;  
END_STRUCT
END_TYPE

